// Mitsubishi GX Works2 project: PLC22_ShitNew22 (2)22נודר   PLC: FX3G

// global labels: Global1
VAR_GLOBAL
  Start_Work_Day AT X007 : BOOL;
  E_Stop AT X005 : BOOL;
  Work_Day_ON AT Y007 : BOOL;
  Inventory_Empty AT M5 : BOOL;
  Gummy_Gum_Value AT D1200 : REAL;
  Is_Prem_Pack AT M0 : BOOL;
END_VAR
VAR_GLOBAL CONSTANT
  K500_Condition : REAL := 500;
  K50_Condition : INT := 500;
  const_5 : REAL := 5;
  const_10 : REAL := 10;
  const_400 : REAL := 400;
END_VAR
VAR_GLOBAL
  Check_Maraz_Type AT X001 : BOOL;
  Check_Maraz_Pinuk AT X001 : BOOL;
  Input_Maraz_Type AT X001 : BOOL;
  Set_Lemon_Amount AT D1300 : REAL;
  Set_Raspberry_Amount AT D1304 : REAL;
  Set_Gummy_Amount AT D1312 : REAL;
  Lemon_Tank_Level AT D1302 : REAL;
  Raspberry_Tank_Level AT D1306 : REAL;
  Gummy_Tank_Level AT D1314 : REAL;
  Set_Stabilizer_Amount AT D1308 : REAL;
  Stabilizer_Tank_Level AT D1310 : REAL;
  Init_Materials AT X001 : BOOL;
  Check_Maraz_Regular AT X001 : BOOL;
END_VAR
VAR_GLOBAL CONSTANT
  const_0 : REAL;
END_VAR
VAR_GLOBAL
  Is_Reg_Pack AT M1 : BOOL;
END_VAR
VAR_GLOBAL CONSTANT
  const_7 : REAL := 7;
END_VAR
VAR_GLOBAL
  Init_Materials_Tanks AT X001 : BOOL;
  Init_Materials_IceCreams AT X001 : BOOL;
END_VAR
VAR_GLOBAL CONSTANT
  const_280 : REAL := 280;
  const_455 : REAL := 455;
  const_105 : REAL := 105;
END_VAR
VAR_GLOBAL
  Init_Materials_And_Maraz_Type AT X001 : BOOL;
  Analog_Input1 AT D8280 : INT;
  Inventory_Check AT X001 : BOOL;
  Init_Materials_And_Analog_Input AT X001 : BOOL;
END_VAR
VAR_GLOBAL CONSTANT
  const_665 : REAL := 665;
  const_210 : REAL := 210;
  const_385 : REAL := 385;
  const_70 : REAL := 70;
  const_28 : REAL := 28;
END_VAR
VAR_GLOBAL
  Start_Production AT X001 : BOOL;
END_VAR
VAR_GLOBAL CONSTANT
  K_50 : INT := 50;
  Time_Limit1 : INT := 50;
END_VAR
VAR_GLOBAL
  TC1 AT TC1 : BOOL;
  P_Timer AT TC1 : BOOL;
  Process_Complete AT TS1 : BOOL;
  Run_Indicator AT Y000 : BOOL;
  Total_Lemon_Produced AT D1316 : REAL;
  Total_Raspberry_Produced AT D1318 : REAL;
END_VAR
VAR_GLOBAL CONSTANT
  const_560 : REAL := 560;
  const_140 : REAL;
  const_560_lemon : REAL := 560;
  const_140_Stabilizer : REAL := 140;
  const_105_Lemon : REAL := 105;
  const_70_Stabilizer : REAL := 70;
  const_280_Raspberry : REAL := 280;
  const_420_Lemon : REAL := 420;
  const_35_Lemon : REAL := 35;
  const_35_Stabilizer : REAL := 35;
  const_385_Raspberry : REAL := 385;
END_VAR
VAR_GLOBAL
  refill_Blocker AT M3 : BOOL;
  Init_Analog_Input AT X001 : BOOL;
  Final_Input AT M66 : BOOL;
  TC2 AT TC2 : BOOL;
  Cool_Timer AT TC2 : BOOL;
  Cooling_Complete AT TS2 : BOOL;
END_VAR
VAR_GLOBAL CONSTANT
  K_80 : INT := 80;
  Time_Limit2 : INT := 80;
END_VAR
VAR_GLOBAL
  Cool_Indicator AT Y002 : BOOL;
  Is_Cold AT X003 : BOOL;
  Cooled_Total_Lemon_Produced AT D1320 : REAL;
  Cooled_Total_Raspberry_Produced AT D1322 : REAL;
  Mix_Tank AT D1324 : REAL;
  Mix_Indicator_5 AT Y005 : BOOL;
  Mix_Indicator_6 AT Y006 : BOOL;
  Cooled_Lemon_Complete AT M6 : BOOL;
  Cooled_Raspberry_Complete AT M7 : BOOL;
  Blink_Mix AT M8 : BOOL;
  TC3 AT TC3 : BOOL;
  Mix_Timer1 AT TC3 : BOOL;
  Mix_Complete1 AT TS3 : BOOL;
END_VAR
VAR_GLOBAL CONSTANT
  K_30 : INT := 30;
  Time_Limit3 : INT := 30;
END_VAR
VAR_GLOBAL
  TC4 AT TC4 : BOOL;
  Mix_Timer2 AT TC4 : BOOL;
  Mix_Complete2 AT TS4 : BOOL;
  TC5 AT TC5 : BOOL;
  Mix_Timer3 AT TC5 : BOOL;
  Mix_Complete3 AT TS5 : BOOL;
  TC6 AT TC6 : BOOL;
  Mix_Timer4 AT TC6 : BOOL;
  Mix_Complete4 AT TS6 : BOOL;
END_VAR
VAR_GLOBAL CONSTANT
  K_10 : INT := 10;
END_VAR
VAR_GLOBAL
  Mix_Process_Complete AT M9 : BOOL;
END_VAR
VAR_GLOBAL CONSTANT
  const_1 : REAL := 1;
END_VAR
VAR_GLOBAL
  Analog_output AT D8282 : INT;
  Batch_Manufacture_Complete AT M10 : BOOL;
  Counter_units AT D1326 : REAL;
  Check AT M20 : BOOL;
  Cooling_Process_Complete AT M67 : BOOL;
  RST_Batch AT X001 : BOOL;
END_VAR
VAR_GLOBAL CONSTANT
  const_40 : REAL := 40;
END_VAR

// task Task_01 (event TRUE, interval 0, priority 31): POU_01

PROGRAM POU_01
(* structured ladder/FBD written out as ST: instructions are called as NAME(EN, inputs, outputs); _pN, _eN, _tN stand for wires *)
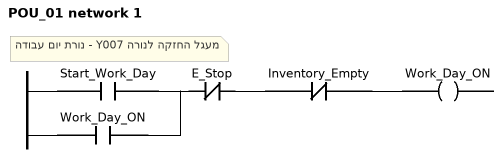
(* network 1 *)
(* מעגל החזקה לנורה Y007 - נורת יום עבודה *)
Work_Day_ON := ((Start_Work_Day OR Work_Day_ON) AND NOT E_Stop) AND NOT Inventory_Empty;
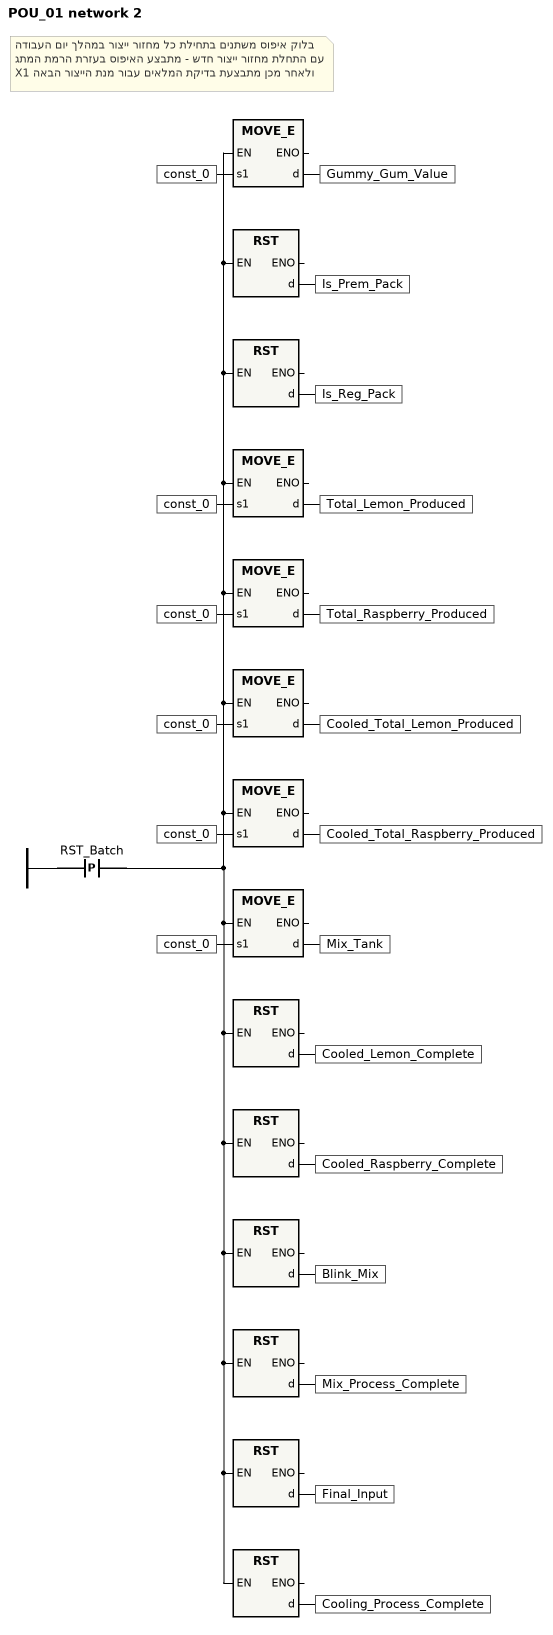
(* network 2 *)
(* בלוק איפוס משתנים בתחילת כל מחזור ייצור במהלך יום העבודה / עם התחלת מחזור ייצור חדש - מתבצע האיפוס בעזרת הרמת המתג X1 ולאחר מכן מתבצעת בדיקת המלאים עבור מנת הייצור הבאה *)
_p1 := LDP(TRUE, RST_Batch);
MOVE_E(_p1, const_0, Gummy_Gum_Value);
RST(_p1, Is_Prem_Pack);
RST(_p1, Is_Reg_Pack);
MOVE_E(_p1, const_0, Total_Lemon_Produced);
MOVE_E(_p1, const_0, Total_Raspberry_Produced);
MOVE_E(_p1, const_0, Cooled_Total_Lemon_Produced);
MOVE_E(_p1, const_0, Cooled_Total_Raspberry_Produced);
MOVE_E(_p1, const_0, Mix_Tank);
RST(_p1, Cooled_Lemon_Complete);
RST(_p1, Cooled_Raspberry_Complete);
RST(_p1, Blink_Mix);
RST(_p1, Mix_Process_Complete);
RST(_p1, Final_Input);
RST(_p1, Cooling_Process_Complete);
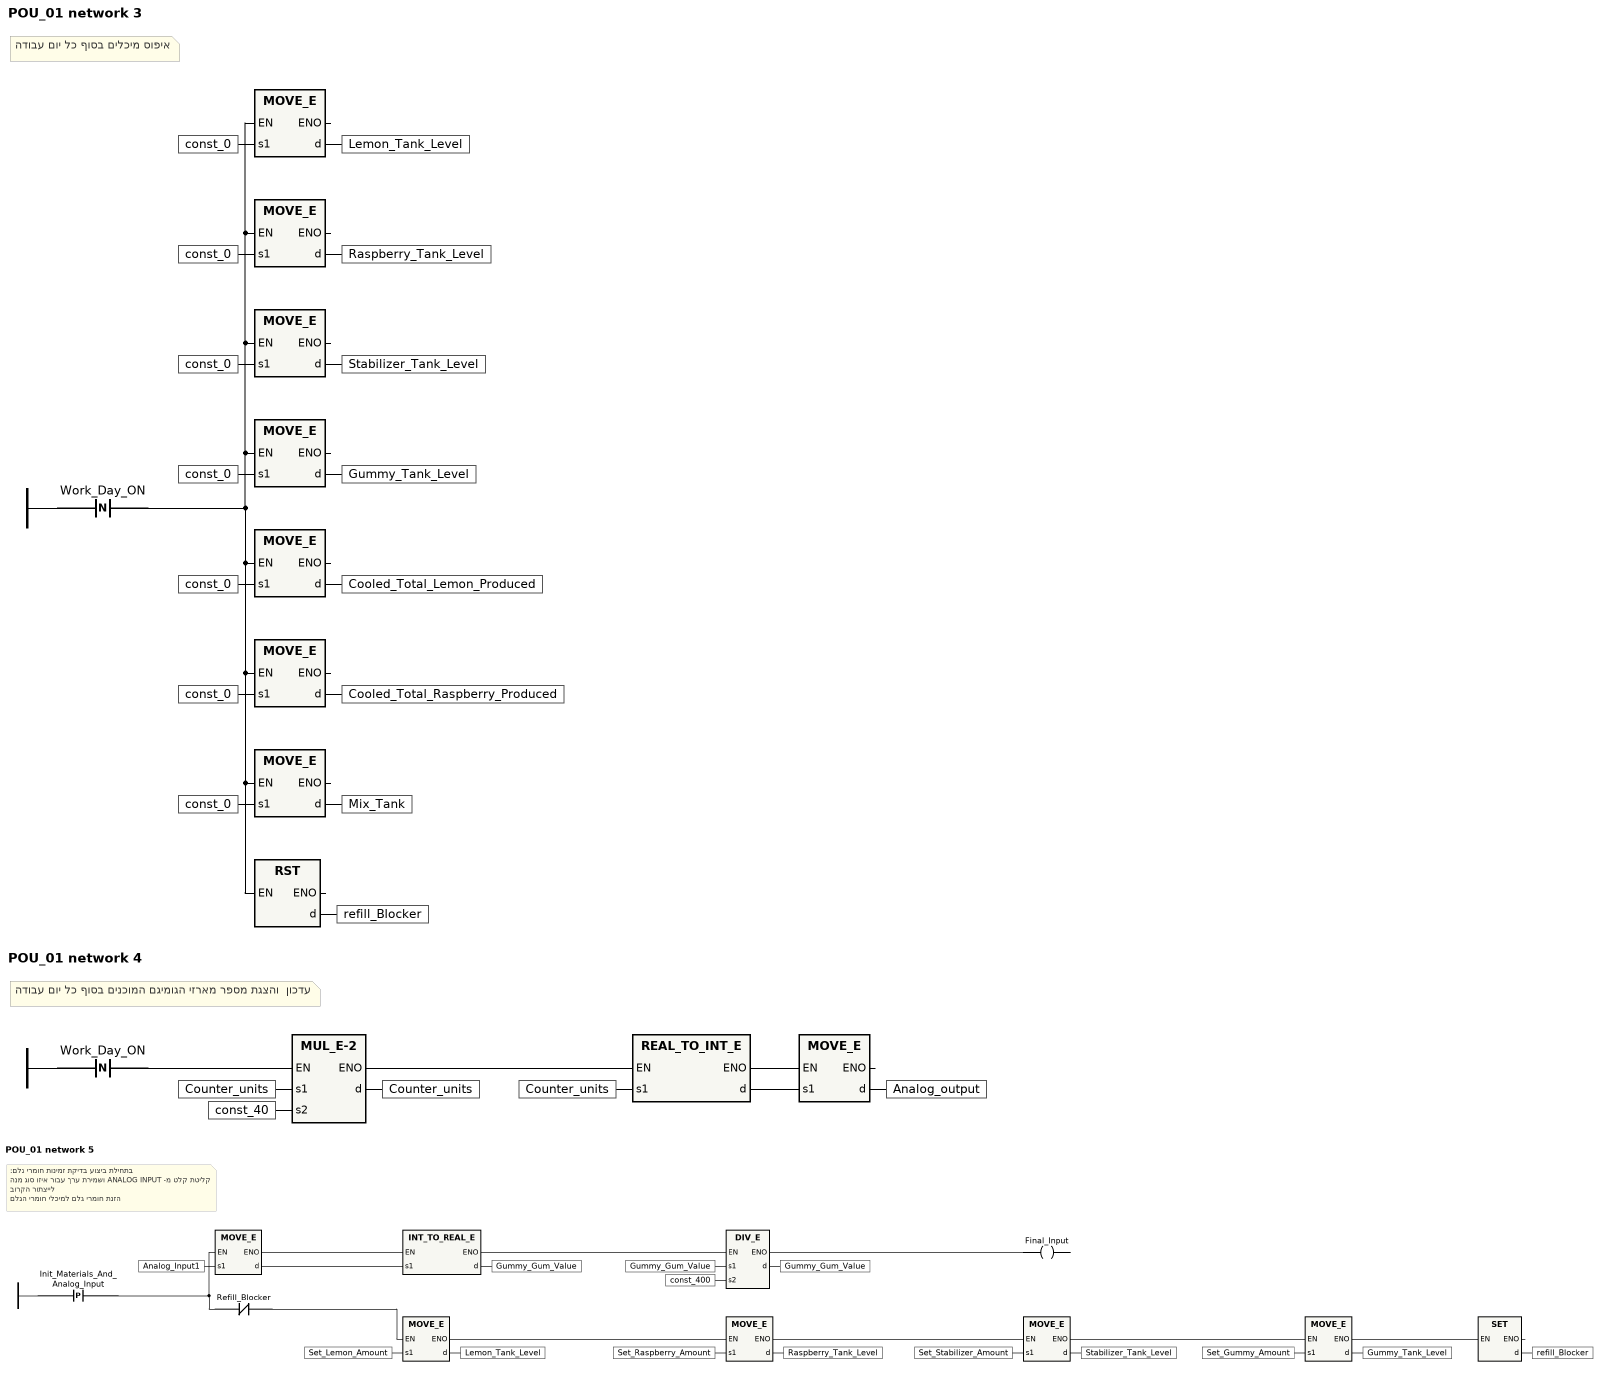
(* network 3 *)
(* איפוס מיכלים בסוף כל יום עבודה *)
_p1 := LDF(TRUE, Work_Day_ON);
MOVE_E(_p1, const_0, Lemon_Tank_Level);
MOVE_E(_p1, const_0, Raspberry_Tank_Level);
MOVE_E(_p1, const_0, Stabilizer_Tank_Level);
MOVE_E(_p1, const_0, Gummy_Tank_Level);
MOVE_E(_p1, const_0, Cooled_Total_Lemon_Produced);
MOVE_E(_p1, const_0, Cooled_Total_Raspberry_Produced);
MOVE_E(_p1, const_0, Mix_Tank);
RST(_p1, refill_Blocker);
(* network 4 *)
(* עדכון  והצגת מספר מארזי הגומיגם המוכנים בסוף כל יום עבודה *)
_e1 := MUL_E(LDF(TRUE, Work_Day_ON), Counter_units, const_40, Counter_units);
_e3 := REAL_TO_INT_E(_e1, Counter_units, _t2);
MOVE_E(_e3, _t2, Analog_output);
(* network 5 *)
(* בתחילת ביצוע בדיקת זמינות חומרי גלם: /  / קליטת קלט מ- ANALOG INPUT ושמירת ערך עבור איזו סוג מנה לייצתור הקרוב /  / הזנת חומרי גלם למיכלי חומרי הגלם *)
_p1 := LDP(TRUE, Init_Materials_And_Analog_Input);
_e3 := MOVE_E(_p1, Analog_Input1, _t2);
_e4 := INT_TO_REAL_E(_e3, _t2, Gummy_Gum_Value);
_e5 := DIV_E(_e4, Gummy_Gum_Value, const_400, Gummy_Gum_Value);
Final_Input := _e5;
_e6 := MOVE_E(_p1 AND NOT Refill_Blocker, Set_Lemon_Amount, Lemon_Tank_Level);
_e7 := MOVE_E(_e6, Set_Raspberry_Amount, Raspberry_Tank_Level);
_e8 := MOVE_E(_e7, Set_Stabilizer_Amount, Stabilizer_Tank_Level);
_e9 := MOVE_E(_e8, Set_Gummy_Amount, Gummy_Tank_Level);
SET(_e9, refill_Blocker);
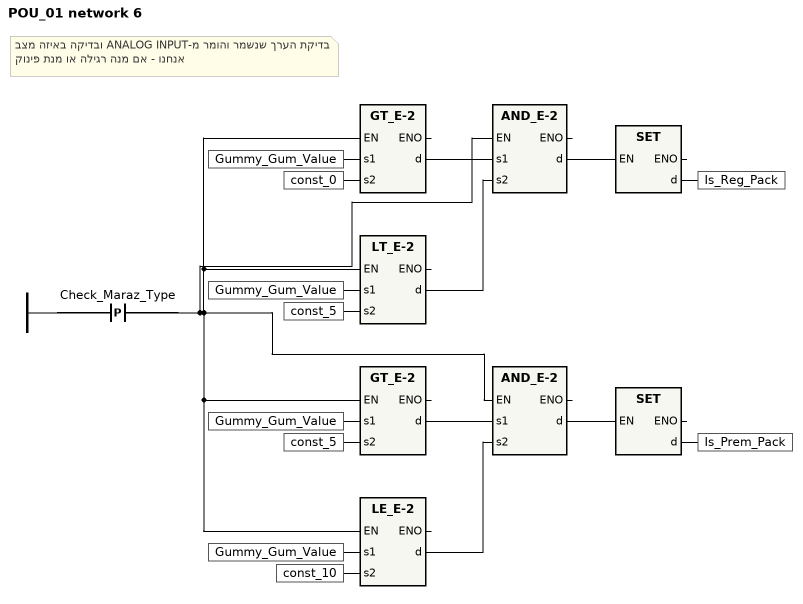
(* network 6 *)
(* בדיקת הערך שנשמר והומר מ-ANALOG INPUT ובדיקה באיזה מצב אנחנו - אם מנה רגילה או מנת פינוק *)
_p1 := LDP(TRUE, Check_Maraz_Type);
GT_E(_p1, Gummy_Gum_Value, const_0, _t2);
LT_E(_p1, Gummy_Gum_Value, const_5, _t3);
AND_E(_p1, _t2, _t3, _t4);
SET(_t4, Is_Reg_Pack);
GT_E(_p1, Gummy_Gum_Value, const_5, _t5);
LE_E(_p1, Gummy_Gum_Value, const_10, _t6);
AND_E(_p1, _t5, _t6, _t7);
SET(_t7, Is_Prem_Pack);
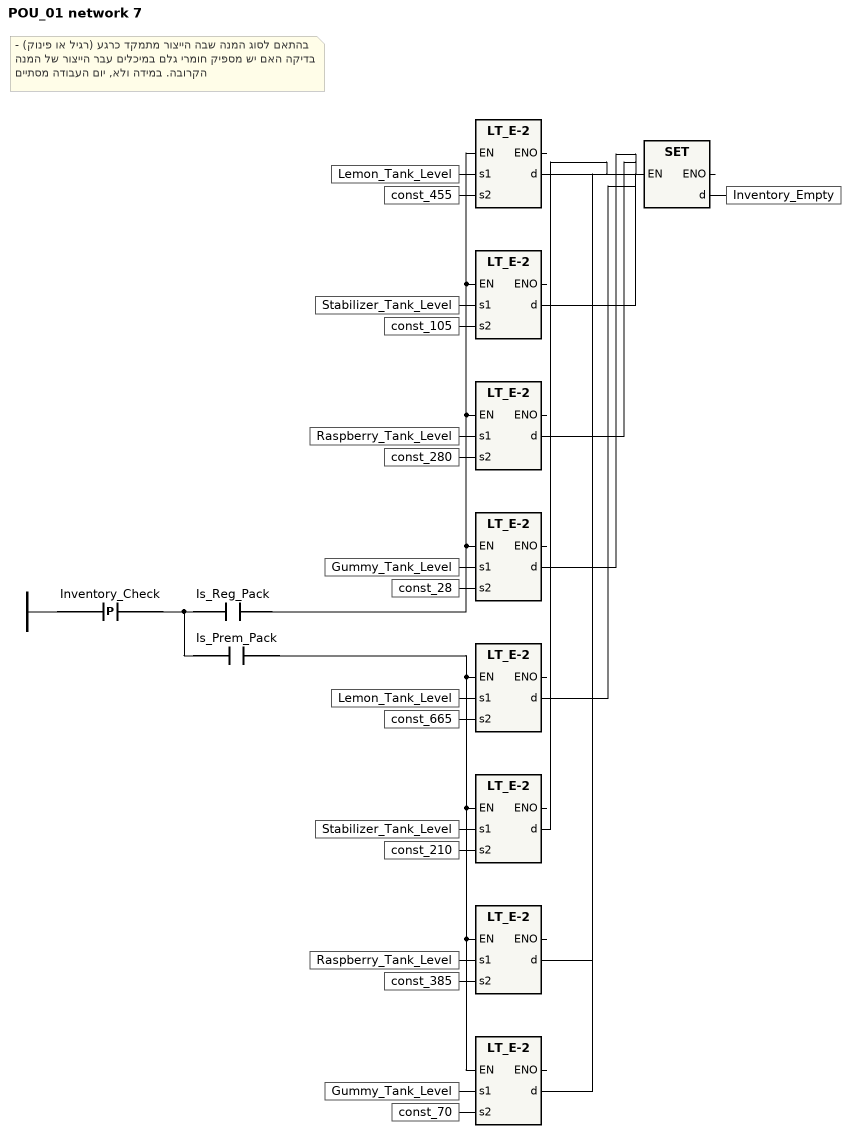
(* network 7 *)
(* בהתאם לסוג המנה שבה הייצור מתמקד כרגע (רגיל או פינוק) - בדיקה האם יש מספיק חומרי גלם במיכלים עבר הייצור של המנה הקרובה. במידה ולא, יום העבודה מסתיים *)
_p1 := LDP(TRUE, Inventory_Check);
_p2 := _p1 AND Is_Reg_Pack;
LT_E(_p2, Lemon_Tank_Level, const_455, _t3);
LT_E(_p2, Stabilizer_Tank_Level, const_105, _t4);
LT_E(_p2, Raspberry_Tank_Level, const_280, _t5);
LT_E(_p2, Gummy_Tank_Level, const_28, _t6);
_p7 := _p1 AND Is_Prem_Pack;
LT_E(_p7, Lemon_Tank_Level, const_665, _t8);
LT_E(_p7, Stabilizer_Tank_Level, const_210, _t9);
LT_E(_p7, Raspberry_Tank_Level, const_385, _t10);
LT_E(_p7, Gummy_Tank_Level, const_70, _t11);
SET(_t3 OR _t4 OR _t5 OR _t6 OR _t8 OR _t9 OR _t10 OR _t11, Inventory_Empty);
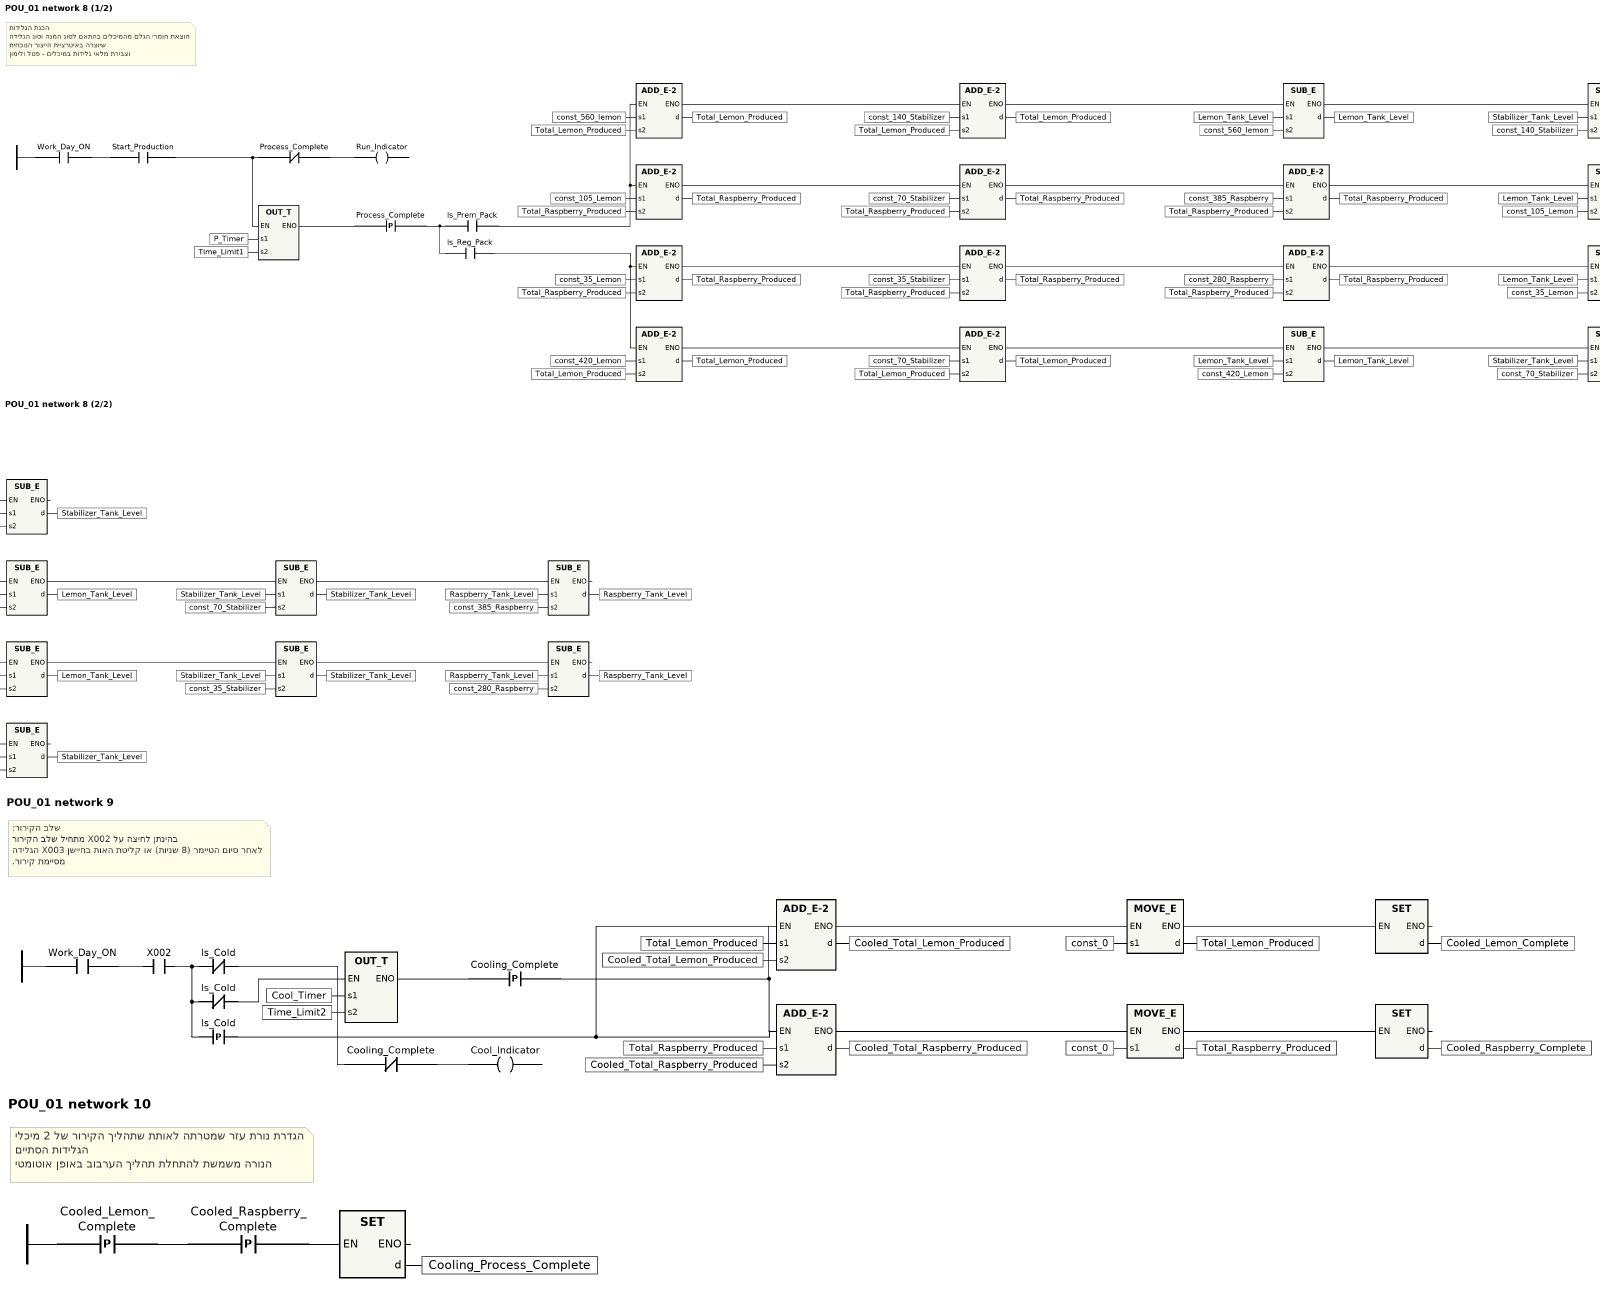
(* network 8 *)
(* הכנת הגלידות / הוצאת חומרי הגלם מהמיכלים בהתאם לסוג המנה וסוג הגלידה שיוצרה באיטרציית הייצור הנוכחית / וצבירת מלאי גלידות במיכלים - פטל ולימון *)
_p1 := Work_Day_ON AND Start_Production;
_e2 := OUT_T(_p1, P_Timer, Time_Limit1);
_p3 := _e2 AND LDP(TRUE, Process_Complete);
_p4 := _p3 AND Is_Prem_Pack;
_e5 := ADD_E(_p4, const_560_lemon, Total_Lemon_Produced, Total_Lemon_Produced);
_e6 := ADD_E(_e5, const_140_Stabilizer, Total_Lemon_Produced, Total_Lemon_Produced);
_e7 := SUB_E(_e6, Lemon_Tank_Level, const_560_lemon, Lemon_Tank_Level);
SUB_E(_e7, Stabilizer_Tank_Level, const_140_Stabilizer, Stabilizer_Tank_Level);
Run_Indicator := _p1 AND NOT Process_Complete;
_e8 := ADD_E(_p4, const_105_Lemon, Total_Raspberry_Produced, Total_Raspberry_Produced);
_e9 := ADD_E(_e8, const_70_Stabilizer, Total_Raspberry_Produced, Total_Raspberry_Produced);
_e10 := ADD_E(_e9, const_385_Raspberry, Total_Raspberry_Produced, Total_Raspberry_Produced);
_e11 := SUB_E(_e10, Lemon_Tank_Level, const_105_Lemon, Lemon_Tank_Level);
_e12 := SUB_E(_e11, Stabilizer_Tank_Level, const_70_Stabilizer, Stabilizer_Tank_Level);
SUB_E(_e12, Raspberry_Tank_Level, const_385_Raspberry, Raspberry_Tank_Level);
_p13 := _p3 AND Is_Reg_Pack;
_e14 := ADD_E(_p13, const_420_Lemon, Total_Lemon_Produced, Total_Lemon_Produced);
_e15 := ADD_E(_e14, const_70_Stabilizer, Total_Lemon_Produced, Total_Lemon_Produced);
_e16 := SUB_E(_e15, Lemon_Tank_Level, const_420_Lemon, Lemon_Tank_Level);
SUB_E(_e16, Stabilizer_Tank_Level, const_70_Stabilizer, Stabilizer_Tank_Level);
_e17 := ADD_E(_p13, const_35_Lemon, Total_Raspberry_Produced, Total_Raspberry_Produced);
_e18 := ADD_E(_e17, const_35_Stabilizer, Total_Raspberry_Produced, Total_Raspberry_Produced);
_e19 := ADD_E(_e18, const_280_Raspberry, Total_Raspberry_Produced, Total_Raspberry_Produced);
_e20 := SUB_E(_e19, Lemon_Tank_Level, const_35_Lemon, Lemon_Tank_Level);
_e21 := SUB_E(_e20, Stabilizer_Tank_Level, const_35_Stabilizer, Stabilizer_Tank_Level);
SUB_E(_e21, Raspberry_Tank_Level, const_280_Raspberry, Raspberry_Tank_Level);
(* network 9 *)
(* שלב הקירור: / בהינתן לחיצה על X002 מתחיל שלב הקירור / לאחר סיום הטיימר (8 שניות) או קליטת האות בחיישן X003 הגלידה מסיימת קירור. *)
_p1 := Work_Day_ON AND X002;
Cool_Indicator := _p1 AND NOT Is_Cold AND NOT Cooling_Complete;
_e2 := OUT_T(_p1 AND NOT Is_Cold, Cool_Timer, Time_Limit2);
_p3 := (_e2 AND LDP(TRUE, Cooling_Complete)) OR (_p1 AND LDP(TRUE, Is_Cold));
_e4 := ADD_E(_p3, Total_Lemon_Produced, Cooled_Total_Lemon_Produced, Cooled_Total_Lemon_Produced);
_e5 := MOVE_E(_e4, const_0, Total_Lemon_Produced);
SET(_e5, Cooled_Lemon_Complete);
_e6 := ADD_E(_p3, Total_Raspberry_Produced, Cooled_Total_Raspberry_Produced, Cooled_Total_Raspberry_Produced);
_e7 := MOVE_E(_e6, const_0, Total_Raspberry_Produced);
SET(_e7, Cooled_Raspberry_Complete);
(* network 10 *)
(* הגדרת נורת עזר שמטרתה לאותת שתהליך הקירור של 2 מיכלי הגלידות הסתיים / הנורה משמשת להתחלת תהליך הערבוב באופן אוטומטי *)
SET(LDP(TRUE, Cooled_Lemon_Complete) AND LDP(TRUE, Cooled_Raspberry_Complete), Cooling_Process_Complete);
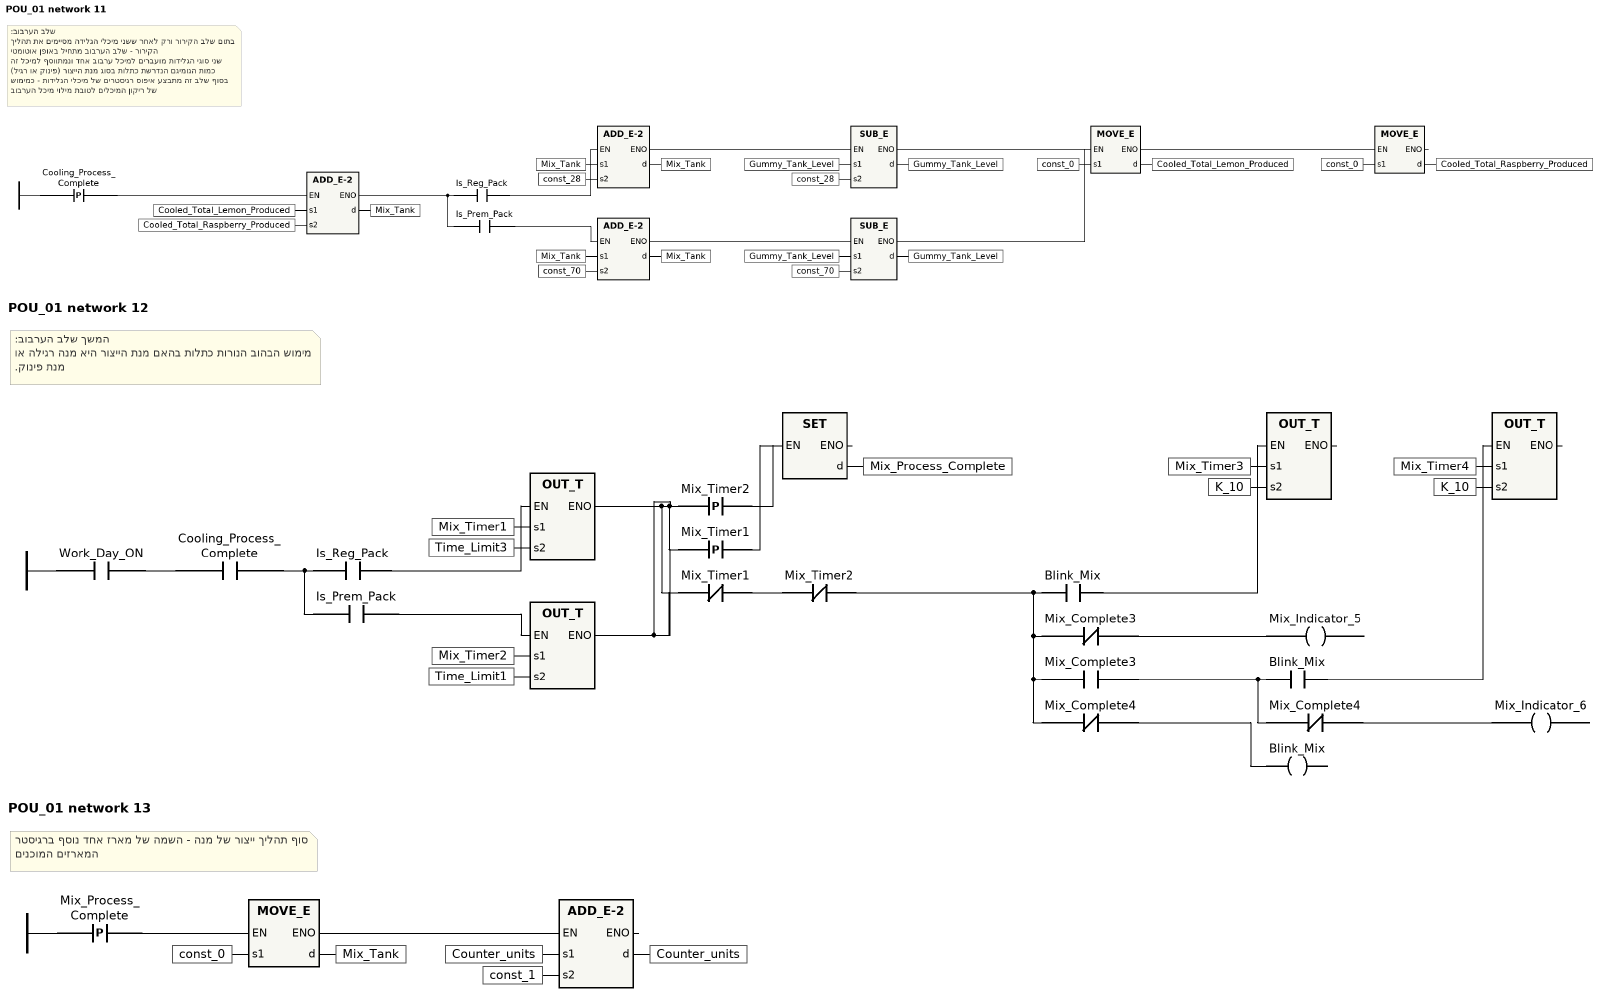
(* network 11 *)
(* שלב הערבוב: / בתום שלב הקירור ורק לאחר ששני מיכלי הגלידה מסיימים את תהליך הקירור - שלב הערבוב מתחיל באופן אוטומטי / שני סוגי הגלידות מועברים למיכל ערבוב אחד ונמתווסף למיכל זה כמות הגומיגם הנדרשת כתלות בסוג מנת הייצור (פינוק או רגיל) / בסוף שלב זה מתבצע איפוס רגיסטרים של מיכלי הגלידות - כמימוש של ריקון המיכלים לטובת מילוי מיכל הערבוב *)
_e1 := ADD_E(LDP(TRUE, Cooling_Process_Complete), Cooled_Total_Lemon_Produced, Cooled_Total_Raspberry_Produced, Mix_Tank);
_e2 := ADD_E(_e1 AND Is_Reg_Pack, Mix_Tank, const_28, Mix_Tank);
_e3 := SUB_E(_e2, Gummy_Tank_Level, const_28, Gummy_Tank_Level);
_e4 := ADD_E(_e1 AND Is_Prem_Pack, Mix_Tank, const_70, Mix_Tank);
_e5 := SUB_E(_e4, Gummy_Tank_Level, const_70, Gummy_Tank_Level);
_e6 := MOVE_E(_e3 OR _e5, const_0, Cooled_Total_Lemon_Produced);
MOVE_E(_e6, const_0, Cooled_Total_Raspberry_Produced);
(* network 12 *)
(* המשך שלב הערבוב: / מימוש הבהוב הנורות כתלות בהאם מנת הייצור היא מנה רגילה או מנת פינוק. *)
_p1 := Work_Day_ON AND Cooling_Process_Complete;
_e2 := OUT_T(_p1 AND Is_Reg_Pack, Mix_Timer1, Time_Limit3);
_e3 := OUT_T(_p1 AND Is_Prem_Pack, Mix_Timer2, Time_Limit1);
_p4 := _e2 OR _e3;
SET((_p4 AND LDP(TRUE, Mix_Timer2)) OR (_p4 AND LDP(TRUE, Mix_Timer1)), Mix_Process_Complete);
_p5 := _p4 AND NOT Mix_Timer1 AND NOT Mix_Timer2;
OUT_T(_p5 AND Blink_Mix, Mix_Timer3, K_10);
Mix_Indicator_5 := _p5 AND NOT Mix_Complete3;
_p6 := _p5 AND Mix_Complete3;
OUT_T(_p6 AND Blink_Mix, Mix_Timer4, K_10);
Mix_Indicator_6 := _p6 AND NOT Mix_Complete4;
Blink_Mix := _p5 AND NOT Mix_Complete4;
(* network 13 *)
(* סוף תהליך ייצור של מנה - השמה של מארז אחד נוסף ברגיסטר המארזים המוכנים *)
_e1 := MOVE_E(LDP(TRUE, Mix_Process_Complete), const_0, Mix_Tank);
ADD_E(_e1, Counter_units, const_1, Counter_units);
END_PROGRAM
